FUNCTION_BLOCK FB_SLITS
VAR_IN_OUT

END_VAR
VAR_INPUT

END_VAR
VAR_OUTPUT
END_VAR
VAR



END_VAR

ACTION ACT_BLOCK:

END_ACTION

ACTION ACT_CalculatePositions:

END_ACTION

END_FUNCTION_BLOCK

(* stored: Version 1.1.0.1, ProductVersion 3.1.4022.18
   POU FB_SLITS: Id {e16e0f37-b04b-4e2b-a3f3-e910fdc91095}, SpecialFunc None
   Action ACT_BLOCK: Id {c3009c9d-9569-4a50-a724-b9e8e026c19a}
   Action ACT_CalculatePositions: Id {725e398a-6162-44d6-8bb7-0ca8a4916528} *)
